// TwinCAT 3 PLC project TcComposite
// Title: TcComposite
// Company: Krystian Lis
// Author: Krystian Lis
// ProjectVersion: 0.001
// ProgramVersion: 3.1.4023.0
// libraries:
//   Tc2_Standard, * (Beckhoff Automation GmbH)
//   Tc2_System, * (Beckhoff Automation GmbH)
//   Tc2_Utilities, * (Beckhoff Automation GmbH)
//   Tc3_Module, * (Beckhoff Automation GmbH)
//   VisuDialogs, * (System)
// project tree:
//   DUTs/TestSt/ ST_PID.TcDUT
//   / GlobalTextList.TcGTLO, PlcTask.TcTTO, Visualization Manager.TcVMO (not stored), VISU_TASK.TcTTO
//   GVLs/ GVL_Data.TcGVL, G.TcGVL, GVL_Sys.TcGVL
//   POUs/Loggers/Functions/ F_Log.TcPOU, UINT_TO_ZEROSTRING.TcPOU
//   POUs/Loggers/ LogList.TcPOU
//   POUs/Objects/Abstracts/Base/ I_BoolPub.TcIO, I_BoolSub.TcIO
//   POUs/Objects/Abstracts/ I_Object.TcIO, I_SYS_COMP_Object.TcIO, Object.TcPOU
//   POUs/Objects/Base/ BoolSub.TcPOU, BoolPub.TcPOU
//   POUs/Objects/Composite/ Timer.TcPOU
//   POUs/Objects/ObjectList/Functions/ F_Get_Parent_Path.TcPOU
//   POUs/Objects/ObjectList/ _SYS_COMP_FirstObject.TcPOU, _SYS_COMP_.TcPOU
//   POUs/Objects/TestObj/ A.TcPOU, B.TcPOU, C.TcPOU
//   POUs/Params/Abstracts/ BaseParam.TcPOU, I_Param.TcIO
//   POUs/Params/ BoolParam.TcPOU, DintParam.TcPOU, RealParam.TcPOU, TimeParam.TcPOU, UdintParam.TcPOU
//   POUs/Params/Functions/ F_Change_Param.TcPOU, F_IObject_TO_IParam.TcPOU
//   POUs/Programs/ MAIN.TcPOU
//   POUs/System/Abstracts/ I_Blank.TcIO, I_Label.TcIO, Label.TcPOU
//   VISUs/ LandingPage.TcVIS, ObjectBrowser.TcVIS, ParamDialog.TcVIS, LogVisu.TcVIS, VisuComments.TcPOU
// real-time tasks:
//   TASK PlcTask: cycle T#10ms, priority 20, ADS port 350
//   TASK VISU_TASK: cycle T#200000us, priority 30, ADS port 351

CONFIGURATION TcComposite
    RESOURCE PLC ON TwinCAT3
        TASK PlcTask(INTERVAL := T#10ms, PRIORITY := 20);
        TASK VISU_TASK(INTERVAL := T#200000us, PRIORITY := 30);
        PROGRAM MAIN WITH PlcTask : MAIN;
        PROGRAM VisuElems_Visu_Prg WITH VISU_TASK : VisuElems.Visu_Prg;
    END_RESOURCE
END_CONFIGURATION

// ---- DUTs/TestSt/ST_PID.TcDUT
//Test structure
//Check if object can ignore struct types when trying to find its parent
// Parent
//	-Struct
//	--Child 1
//	--Child 2
//	--Child 3
//Struct should be ignored and child should be added directly to the parent


TYPE ST_PID :
STRUCT
	p: RealParam;
	i: RealParam;
	d: RealParam;
END_STRUCT
END_TYPE

// ---- GVLs/GVL_Data.TcGVL
//Test GVL
{attribute 'qualified_only'}
VAR_GLOBAL
END_VAR

// ---- GVLs/G.TcGVL
//Test GVL
{attribute 'qualified_only'}
VAR_GLOBAL
A1: A;
A2: A;
A3: A;
END_VAR

// ---- GVLs/GVL_Sys.TcGVL
//Test GVL
{attribute 'qualified_only'}
VAR_GLOBAL
END_VAR

// ---- POUs/Objects/Abstracts/Base/I_BoolPub.TcIO
INTERFACE I_BoolPub EXTENDS I_SYS_COMP_Object

//Work in progress

METHOD Attach_Sub
VAR_INPUT
	IObject: I_SYS_COMP_Object;
END_VAR
END_METHOD

PROPERTY Get : BOOL
GET
END_GET
END_PROPERTY

METHOD Remove_Sub
VAR_INPUT
	IObject: I_SYS_COMP_Object;
END_VAR
END_METHOD

END_INTERFACE

// ---- POUs/Objects/Abstracts/Base/I_BoolSub.TcIO
INTERFACE I_BoolSub EXTENDS I_SYS_COMP_Object

//Work in progress

METHOD Attach_Pub
VAR_INPUT
	IObject: I_SYS_COMP_Object;
END_VAR
END_METHOD

METHOD Remove_Pub
VAR_INPUT
	IObject: I_SYS_COMP_Object;
END_VAR
END_METHOD

PROPERTY Set : BOOL
SET
END_SET
END_PROPERTY

END_INTERFACE

// ---- POUs/Objects/Abstracts/I_Object.TcIO
INTERFACE I_Object EXTENDS I_Label

//I_SYS_COMP_Object facade

METHOD Get_Child : I_Object
VAR_INPUT
	name: STRING;
END_VAR
END_METHOD

METHOD Get_Parent : I_Object
VAR_INPUT
END_VAR
END_METHOD

METHOD Refresh
VAR_INPUT
END_VAR
END_METHOD

END_INTERFACE

// ---- POUs/Objects/Abstracts/I_SYS_COMP_Object.TcIO
INTERFACE I_SYS_COMP_Object EXTENDS I_Label

//System interface, shouldn't be modified

METHOD _SYS_COMP_Add_Child_
VAR_INPUT
	IObject: I_SYS_COMP_Object;
END_VAR
END_METHOD

METHOD _SYS_COMP_Get_Child : I_SYS_COMP_Object
VAR_INPUT
	name: STRING;
END_VAR
END_METHOD

METHOD _SYS_COMP_Get_Object : I_SYS_COMP_Object
VAR_INPUT
	parent_name: STRING;
	name: STRING;
END_VAR
END_METHOD

PROPERTY _SYS_COMP_last_child : I_SYS_COMP_Object
GET
END_GET
END_PROPERTY

PROPERTY _SYS_COMP_next_object : I_SYS_COMP_Object
GET
END_GET
SET
END_SET
END_PROPERTY

PROPERTY _SYS_COMP_parent : I_SYS_COMP_Object
GET
END_GET
SET
END_SET
END_PROPERTY

PROPERTY _SYS_COMP_prev_object : I_SYS_COMP_Object
GET
END_GET
SET
END_SET
END_PROPERTY

METHOD _SYS_COMP_Remove_Child_
VAR_INPUT
	IObject: I_SYS_COMP_Object;
END_VAR
END_METHOD

END_INTERFACE

// ---- POUs/Params/Abstracts/I_Param.TcIO
INTERFACE I_Param EXTENDS I_Label

METHOD Change_Param
VAR_INPUT
	value: STRING;
END_VAR
END_METHOD

PROPERTY display : STRING
GET
END_GET
END_PROPERTY

END_INTERFACE

// ---- POUs/System/Abstracts/I_Blank.TcIO
INTERFACE I_Blank EXTENDS __SYSTEM.IQueryInterface

END_INTERFACE

// ---- POUs/System/Abstracts/I_Label.TcIO
INTERFACE I_Label EXTENDS I_Blank

PROPERTY name : STRING
GET
END_GET
END_PROPERTY

END_INTERFACE

// ---- POUs/Programs/MAIN.TcPOU
PROGRAM MAIN
VAR
	rParam: I_Object;

	_init: BOOL;
END_VAR

IF NOT _init THEN
	
	F_Change_Param(
		G.A1.Get_Child('B1').Get_Child('tB'),
		'TRUE');
		
	rParam := G.A1.Get_Child('C1').Get_Child('tR');
	F_Change_Param(rParam, '0.7');

	
	_init := TRUE;
END_IF

END_PROGRAM

// ---- POUs/Params/Functions/F_Change_Param.TcPOU
FUNCTION F_Change_Param : BOOL
VAR_INPUT
	IObject: I_Object;
	value: STRING;
END_VAR
VAR
	_IParam: I_Param;
	_interface_match: BOOL;
END_VAR

//Used to safely change param of unknown object. If object doesn't contain I_Param
//or if it is 0 then it won't work.

_interface_match := __QUERYINTERFACE(IObject, _IParam);
IF _interface_match THEN
	_IParam.Change_Param(value);
END_IF

F_Change_Param := _interface_match;

END_FUNCTION

// ---- POUs/Objects/TestObj/A.TcPOU
{attribute 'call_after_init'}
FUNCTION_BLOCK A EXTENDS Object
VAR_INPUT
END_VAR
VAR_OUTPUT
END_VAR
VAR
	B1: B;
	B2: B;
	B3: B;

	tR: RealParam;
END_VAR

END_FUNCTION_BLOCK

// ---- POUs/Objects/Abstracts/Object.TcPOU
FUNCTION_BLOCK ABSTRACT Object EXTENDS Label IMPLEMENTS I_SYS_COMP_Object, I_Object
VAR

	{attribute 'no_copy'}
	{attribute 'no_init'}
	_SYS_COMP_next_object_: I_SYS_COMP_Object;
	
	{attribute 'no_copy'}
	{attribute 'no_init'}
	_SYS_COMP_prev_object_: I_SYS_COMP_Object;
	
	{attribute 'no_copy'}
	{attribute 'no_init'}
	_SYS_COMP_last_child_: I_SYS_COMP_Object;
	
	{attribute 'no_copy'}
	{attribute 'no_init'}
	_SYS_COMP_parent_: I_SYS_COMP_Object;
	
	{attribute 'no_copy'}
	{attribute 'no_init'}
	_SYS_COMP_init_parent_: BOOL;
	
END_VAR

METHOD _SYS_COMP_Add_Child_
VAR_INPUT
	IObject: I_SYS_COMP_Object;
END_VAR
//Remove from current chain and add to parent chain



IF IObject = 0 THEN
	RETURN;
END_IF

IF IObject._SYS_COMP_parent <> 0 THEN
	RETURN;
END_IF

//_SYS_COMP_.Remove_Object(IObject);

F_Log(IObject, 'ADDED TO', THIS^, '', 0);



IObject._SYS_COMP_parent := THIS^;



IF _SYS_COMP_last_child_ = 0 THEN
	_SYS_COMP_last_child_ := IObject;
	//LOG
	RETURN;	
END_IF


IObject._SYS_COMP_prev_object := _SYS_COMP_last_child_;

_SYS_COMP_last_child_._SYS_COMP_next_object := IObject;


_SYS_COMP_last_child_ := IObject;
END_METHOD

METHOD _SYS_COMP_Find_Parent_
VAR
	_temp_name: STRING;
	_potential_parent: I_SYS_COMP_Object;
END_VAR
// At the initialisation all objects are added to 
// the global list in order parent, child, parent_sibling, parent_sibling_child etc

// At FB_init the object is added to global list and then it's looking for parent
// It first check if previous sybling is its parent, 
// and then if its parent of a parent(of a parent ...)
// if there is no similarity beteen objec and any other object paths,
// the object is not removed from global list.

// Example child name: A.B.C.D.E
// Example previous sibling name: G.A.B
// Example parent name: G.A.B
//Thus the process looks like that:

IF _SYS_COMP_prev_object_ = 0 THEN
	RETURN;
END_IF

//Check if previous sybling has similar path as the object
IF FIND(_name, _SYS_COMP_prev_object_.name) <> 0 THEN
	_temp_name := F_Get_Parent_Path(_name);
	//delete name after last dot and check if it matches previous sybling name
	IF _SYS_COMP_prev_object_.name = _temp_name THEN
		_SYS_COMP_prev_object_._SYS_COMP_Add_Child_(THIS^);
		RETURN;
	END_IF
	
	//proceed deleting dots, if any name match the resulting path then set up the parent
	WHILE TRUE DO
		_temp_name := F_Get_Parent_Path(_temp_name);
		_potential_parent := _SYS_COMP_prev_object._SYS_COMP_Get_Child(_temp_name);

		IF _potential_parent <> _SYS_COMP_prev_object THEN
			_potential_parent._SYS_COMP_Add_Child_(THIS^);
			RETURN;	
		END_IF
		
		// if nothing left from the object path, then the object is part of global list
		IF _temp_name = '' THEN
			RETURN;
		END_IF
	END_WHILE
END_IF
END_METHOD

METHOD _SYS_COMP_Get_Child : I_SYS_COMP_Object
VAR_INPUT
	name: STRING;
END_VAR
VAR
	_IObject: I_SYS_COMP_Object;
END_VAR
//Get system object interface

//Add # at the end. This will ensure that the string value 
//is actually on the end of the path
IF RIGHT(name, 1) <> '#' THEN
	name := CONCAT(name, '#');
END_IF

IF _SYS_COMP_last_child_ <> 0 THEN
	_IObject := _SYS_COMP_last_child_._SYS_COMP_Get_Object(_name, name);
END_IF

//For security reasons this method always returns something,
//Thus if object can't be found, the methods return the THIS object
IF _IObject <> 0 THEN
	_SYS_COMP_Get_Child := _IObject;
ELSE
	_SYS_COMP_Get_Child := THIS^;
END_IF
END_METHOD

METHOD _SYS_COMP_Get_Object : I_SYS_COMP_Object
VAR_INPUT
	parent_name: STRING;
	name: STRING;
END_VAR
VAR
	_temp_name: STRING;
	_IObject: I_SYS_COMP_Object;
	_case: USINT;
END_VAR
_temp_name := CONCAT(_name, '#');

IF parent_name = '#' THEN
	//FIND object ending with name# in any parent
	_case := 1;
END_IF

//Check if object matches the searched name,
//If no check if it contain searched name,
//If yes, check in children,
//If not, go to next sibling

CASE _case OF
	0:
		IF FIND(_temp_name, name) <> 0 THEN
			_SYS_COMP_Get_Object := THIS^;
			RETURN;
		END_IF
		IF FIND(_temp_name, parent_name) <> 0 THEN
			_IObject := _SYS_COMP_Get_Child(name);
			IF _IObject <> 0 AND_THEN _name <> _IObject.name THEN
				_SYS_COMP_Get_Object := _IObject;
				RETURN;
			END_IF
		END_IF
	1:	//FIND object ending with name# in any parent
		IF FIND(_temp_name, name) <> 0 THEN
			_SYS_COMP_Get_Object := THIS^;
			RETURN;	
		ELSE
			_IObject := _SYS_COMP_Get_Child(name);
			IF _IObject <> 0 AND_THEN _name <> _IObject.name THEN
				_SYS_COMP_Get_Object := _IObject;
				RETURN;
			END_IF
		END_IF
END_CASE


//Got to next sibling
IF _SYS_COMP_prev_object_ <> 0 THEN
	_SYS_COMP_Get_Object := _SYS_COMP_prev_object_._SYS_COMP_Get_Object(parent_name, name);
	RETURN;
END_IF
END_METHOD

PROPERTY _SYS_COMP_last_child : I_SYS_COMP_Object
GET
_SYS_COMP_last_child := _SYS_COMP_last_child_;
END_GET
END_PROPERTY

PROPERTY _SYS_COMP_next_object : I_SYS_COMP_Object
GET
_SYS_COMP_next_object := _SYS_COMP_next_object_;
END_GET
SET
//F_Log(THIS^, 'ATTACH_NEXT', next_object, 'BEFORE', _next_object);
_SYS_COMP_next_object_ := _SYS_COMP_next_object;
END_SET
END_PROPERTY

PROPERTY _SYS_COMP_parent : I_SYS_COMP_Object
GET
_SYS_COMP_parent := _SYS_COMP_parent_;
END_GET
SET
IF NOT _SYS_COMP_init_parent_ THEN
	_SYS_COMP_parent_ := _SYS_COMP_parent;
	_SYS_COMP_init_parent_ := TRUE;
END_IF
END_SET
END_PROPERTY

PROPERTY _SYS_COMP_prev_object : I_SYS_COMP_Object
GET
_SYS_COMP_prev_object := _SYS_COMP_prev_object_;
END_GET
SET
//F_Log(THIS^, 'ATTACH_PREV', prev_object, 'BEFORE', _prev_object);
_SYS_COMP_prev_object_ := _SYS_COMP_prev_object;
END_SET
END_PROPERTY

METHOD _SYS_COMP_Remove_Child_
VAR_INPUT
	IObject: I_SYS_COMP_Object;
END_VAR
IF IObject = 0 THEN
	//LOG
	RETURN;
END_IF

IF _SYS_COMP_last_child_ = 0 THEN
	//LOG
	RETURN;
END_IF

IF IObject._SYS_COMP_parent <> 0 AND_THEN IObject._SYS_COMP_parent.name <> _name THEN
	//LOG
	//Object from different parent
	F_Log(IObject, 'IS NOT CHILD OF', THIS^, '', 0);
	RETURN;
END_IF

F_Log(IObject, 'REMOVED FROM', THIS^, '', 0);

IF IObject._SYS_COMP_next_object = 0 AND IObject._SYS_COMP_prev_object <> 0 THEN
	_SYS_COMP_last_child_ := IObject._SYS_COMP_prev_object;
	_SYS_COMP_last_child_._SYS_COMP_next_object := 0;
	
	_SYS_COMP_last_child_ := 0;
	IObject._SYS_COMP_next_object := 0;
	IObject._SYS_COMP_prev_object := 0;
	//LOG
	RETURN;
END_IF

IF IObject._SYS_COMP_next_object <> 0 AND IObject._SYS_COMP_prev_object <> 0 THEN
	IObject._SYS_COMP_next_object._SYS_COMP_prev_object := IObject._SYS_COMP_prev_object;
	IObject._SYS_COMP_prev_object._SYS_COMP_next_object := IObject._SYS_COMP_next_object;


	IObject._SYS_COMP_next_object := 0;
	IObject._SYS_COMP_prev_object := 0;
	//LOG
	RETURN;
END_IF

IF IObject._SYS_COMP_next_object <> 0 AND IObject._SYS_COMP_prev_object = 0 THEN
	IObject._SYS_COMP_next_object._SYS_COMP_prev_object := 0;

	IObject._SYS_COMP_next_object := 0;
	IObject._SYS_COMP_prev_object := 0;
	//LOG
	RETURN;
END_IF
END_METHOD

METHOD FB_exit : BOOL
VAR_INPUT
	bInCopyCode : BOOL; // if TRUE, the exit method is called for exiting an instance that is copied afterwards (online change).
END_VAR
//_SYS_COMP_.Remove_Object(THIS^);
END_METHOD

METHOD FB_init : BOOL
VAR_INPUT
	bInitRetains : BOOL; // if TRUE, the retain variables are initialized (warm start / cold start)
	bInCopyCode : BOOL;  // if TRUE, the instance afterwards gets moved into the copy code (online change)
END_VAR
_SYS_COMP_.Add_Object(THIS^);
_SYS_COMP_Find_Parent_();
END_METHOD

METHOD Get_Child : I_Object
VAR_INPUT
	name: STRING;
END_VAR
VAR
	IChild: I_Object;
	ISYSChild: I_SYS_COMP_Object;
END_VAR
//Get child facade interface(without all system methods)

ISYSChild := _SYS_COMP_Get_Child(name);

IF __QUERYINTERFACE(ISYSChild, IChild) THEN
	Get_Child := IChild;
ELSE
	Get_Child := THIS^;
END_IF
END_METHOD

METHOD Get_Parent : I_Object
VAR
	IParent : I_Object;
END_VAR
//Get parent facade interface(without all system methods)

IF __QUERYINTERFACE(_SYS_COMP_parent_, IParent) THEN
	Get_Parent := IParent;
ELSE
	Get_Parent := THIS^;
END_IF
END_METHOD

METHOD Refresh
VAR_INPUT
END_VAR
//User code. Called by children
END_METHOD

END_FUNCTION_BLOCK

// ---- POUs/System/Abstracts/Label.TcPOU
{attribute 'reflection'}
FUNCTION_BLOCK ABSTRACT Label IMPLEMENTS I_Label
VAR CONSTANT
END_VAR
VAR_INPUT
END_VAR
VAR
	
	{attribute 'instance-path'} 
    {attribute 'noinit'}
	_sPath: T_MaxString;
	{attribute 'no_copy'}
	_name: T_MaxString;
	
END_VAR

//Base class. Allows to querry instances by their name.

METHOD FB_init : BOOL
VAR_INPUT
	bInitRetains : BOOL; // if TRUE, the retain variables are initialized (warm start / cold start)
	bInCopyCode : BOOL;  // if TRUE, the instance afterwards gets moved into the copy code (online change)
END_VAR
//Update name after each 'New Download'
_name := DELETE(_sPath, FIND(_sPath, '.'), 1);
_name := DELETE(_name, FIND(_name, '.'), 1);
END_METHOD

PROPERTY name : STRING
GET
name := _name;
END_GET
END_PROPERTY

END_FUNCTION_BLOCK

// ---- POUs/Loggers/Functions/F_Log.TcPOU
FUNCTION F_Log : BOOL
VAR_INPUT
	obj_1	: I_SYS_COMP_Object;
	act_1	: STRING(30);
	obj_2	: I_SYS_COMP_Object;
	act_2	: STRING(30);
	obj_3	: I_SYS_COMP_Object;
END_VAR
VAR
	_remaining_spaces: INT;
	_temp_string: T_MAXSTRING := '                                                                                                                                                                                                                                                               ';
	
	_obj_1_name	: STRING(65);
	_obj_2_name	: STRING(65);
	_obj_3_name	: STRING(65);

END_VAR

//This function creates logs regarding any system related events such as
//Add/Remove Child/Parent etc.

IF obj_1 <> 0 THEN
	_obj_1_name := obj_1.name;
END_IF
IF obj_2 <> 0 THEN
	_obj_2_name := obj_2.name;
END_IF
IF obj_3 <> 0 THEN
	_obj_3_name := obj_3.name;
END_IF

_temp_string := INSERT(_temp_string, _obj_1_name, 0);
_temp_string := INSERT(_temp_string, act_1, 64);
_temp_string := INSERT(_temp_string, _obj_2_name, 94);
_temp_string := INSERT(_temp_string, act_2, 159);
_temp_string := INSERT(_temp_string, _obj_3_name, 189);

LogList.AddLog(_temp_string);

END_FUNCTION

// ---- POUs/Loggers/LogList.TcPOU
{attribute 'global_init_slot' := '40001'}
PROGRAM LogList
VAR
	list: ARRAY[1..4000] OF T_MAXSTRING;
	lastlog: UINT := 1;
END_VAR

//Singleton containing logs

METHOD AddLog
VAR_INPUT
	text: T_MAXSTRING;
END_VAR
list[lastLog] := text;
lastLog := lastLog + 1;

IF lastLog = 4001 THEN
	lastLog := 1;
END_IF
END_METHOD

METHOD Print_To_ADS : DINT
VAR
	_counter : UINT := 1;
	_temp_string: T_MAXSTRING;
	_print_string: T_MAXSTRING;
	_error : DINT;
END_VAR
FOR _counter := 1 TO lastlog DO
	_temp_string := UINT_TO_ZEROSTRING(_counter);
	_temp_string := CONCAT(_temp_string, '  ');
	_temp_string := CONCAT(_temp_string, list[_counter]);
	_print_string := _temp_string;
	
	_error := ADSLOGSTR(ADSLOG_MSGTYPE_STRING, _print_string, '');
	
	IF _error <> 0 THEN
		Print_To_ADS := _error;
		RETURN;
	END_IF
END_FOR
END_METHOD

END_PROGRAM

// ---- POUs/Loggers/Functions/UINT_TO_ZEROSTRING.TcPOU
FUNCTION UINT_TO_ZEROSTRING : T_MAXSTRING
VAR_INPUT
	input : UDINT;
END_VAR
VAR
	tempString : T_MAXSTRING;
END_VAR

tempString := TO_STRING(input);
WHILE LEN(tempString) < 4 DO
	tempString := INSERT(tempString, '0', 0);
END_WHILE
UINT_TO_ZEROSTRING := tempString;

END_FUNCTION

// ---- POUs/Objects/ObjectList/Functions/F_Get_Parent_Path.TcPOU
FUNCTION F_Get_Parent_Path : T_MAXSTRING
VAR_INPUT
	child_path: T_MAXSTRING;
END_VAR
VAR
	_output_string: T_MAXSTRING;
	_dot_position: INT;
END_VAR

WHILE TRUE DO
	_dot_position := FIND(child_path, '.');	
	
	IF _dot_position = 0 THEN
		_output_string := DELETE(_output_string, 1, LEN(_output_string));
		F_Get_Parent_Path := _output_string;
		RETURN;
	END_IF
	
	_output_string := CONCAT(_output_string, LEFT(child_path, _dot_position));
		
	child_path := DELETE(child_path, _dot_position, 1);
	

END_WHILE

END_FUNCTION

// ---- POUs/Objects/ObjectList/_SYS_COMP_.TcPOU
{attribute 'global_init_slot' := '40002'}
{attribute 'hide_all_locals'}
PROGRAM _SYS_COMP_
VAR
	_last_in_chain: I_SYS_COMP_Object;
	_object_list: _SYS_COMP_FirstObject;
END_VAR
VAR CONSTANT
	_name : STRING := 'ObjectList';
END_VAR

METHOD Add_Object
VAR_INPUT
	IObject: I_SYS_COMP_Object;
END_VAR
IF IObject = 0 THEN
	//LOG
	RETURN;
END_IF

//Remove_Object(IObject);

F_Log(IObject, 'ADDED TO', _object_list, '', 0);

IF _last_in_chain = 0 THEN
	_last_in_chain := IObject;
	RETURN;
END_IF

_last_in_chain._SYS_COMP_next_object := IObject;
IObject._SYS_COMP_prev_object := _last_in_chain;
_last_in_chain := IObject;
END_METHOD

METHOD Get_Object : I_SYS_COMP_Object
VAR_INPUT
	name: STRING;
END_VAR
VAR
	_IObject	:	I_SYS_COMP_Object;
END_VAR
name := CONCAT(name, '#');
IF _last_in_chain <> 0 THEN
	_IObject := _last_in_chain._SYS_COMP_Get_Object('#', name);
END_IF

IF _IObject <> 0 THEN
	Get_Object := _IObject;
ELSE
	Get_Object := _object_list;
END_IF

//LOG
END_METHOD

PROPERTY object_list : I_SYS_COMP_Object
GET
object_list := _object_list;
END_GET
END_PROPERTY

METHOD Remove_Object
VAR_INPUT
	IObject: I_SYS_COMP_Object;
END_VAR
IF IObject = 0 THEN
	RETURN;
END_IF

IF IObject._SYS_COMP_prev_object = 0 AND IObject._SYS_COMP_next_object = 0 THEN
	RETURN;
END_IF

IF IObject._SYS_COMP_parent <> 0 THEN
	IObject._SYS_COMP_parent._SYS_COMP_Remove_Child_(IObject);
	RETURN;
END_IF

F_Log(IObject, 'REMOVED FROM', _object_list, '', 0);

IF IObject._SYS_COMP_next_object <> 0 AND IObject._SYS_COMP_prev_object <> 0 THEN
	IObject._SYS_COMP_next_object._SYS_COMP_prev_object := IObject._SYS_COMP_prev_object;
	IObject._SYS_COMP_prev_object._SYS_COMP_next_object := IObject._SYS_COMP_next_object;
	
	IObject._SYS_COMP_next_object := 0;
	IObject._SYS_COMP_prev_object := 0;
	
	
	RETURN;
END_IF

IF IObject._SYS_COMP_next_object = 0 AND IObject._SYS_COMP_prev_object <> 0 THEN
	IObject._SYS_COMP_prev_object._SYS_COMP_next_object := 0;
	_last_in_chain := IObject._SYS_COMP_prev_object;
	
	IObject._SYS_COMP_next_object := 0;
	IObject._SYS_COMP_prev_object := 0;

	RETURN;
END_IF

IF IObject._SYS_COMP_next_object <> 0 AND IObject._SYS_COMP_prev_object = 0 THEN
	IObject._SYS_COMP_next_object._SYS_COMP_prev_object := 0;
	
	IObject._SYS_COMP_next_object := 0;
	IObject._SYS_COMP_prev_object := 0;
	
	RETURN;
END_IF

//LOG
END_METHOD

END_PROGRAM

// ---- POUs/Objects/ObjectList/_SYS_COMP_FirstObject.TcPOU
{attribute 'call_after_init'}
FUNCTION_BLOCK FINAL _SYS_COMP_FirstObject EXTENDS Object
VAR_INPUT
END_VAR
VAR_OUTPUT
END_VAR
VAR
END_VAR

//First object in global object list.
//DO NOT DELETE!!!

END_FUNCTION_BLOCK

// ---- POUs/Objects/TestObj/B.TcPOU
{attribute 'call_after_init'}
FUNCTION_BLOCK B EXTENDS Object
VAR_INPUT
END_VAR
VAR_OUTPUT
END_VAR
VAR
	C1: C;
	C2: C;
	C3: C;

	tR: RealParam;
END_VAR

END_FUNCTION_BLOCK

// ---- POUs/Objects/TestObj/C.TcPOU
{attribute 'call_after_init'}
FUNCTION_BLOCK C EXTENDS Object
VAR_INPUT
END_VAR
VAR_OUTPUT
END_VAR
VAR
	tU: UdintParam;
	tT: TimeParam;
	tR: RealParam;
END_VAR

END_FUNCTION_BLOCK

// ---- POUs/Params/UdintParam.TcPOU
{attribute 'call_after_init'}
FUNCTION_BLOCK FINAL UdintParam EXTENDS BaseParam
VAR_INPUT
END_VAR
VAR_OUTPUT
	value: UDINT;
END_VAR
VAR
	
END_VAR

METHOD Change_Param
VAR_INPUT
	value	: STRING;
END_VAR
THIS^.value := STRING_TO_UDINT(value);
_display := UDINT_TO_STRING(THIS^.value);
END_METHOD

METHOD Quick_Change
VAR_INPUT
	value: UDINT;
END_VAR
THIS^.value := value;
_display := UDINT_TO_STRING(THIS^.value);
END_METHOD

END_FUNCTION_BLOCK

// ---- POUs/Params/Abstracts/BaseParam.TcPOU
FUNCTION_BLOCK ABSTRACT BaseParam EXTENDS Object IMPLEMENTS I_Param
VAR
	_display: STRING := '0';
END_VAR

//Base Param object.
// _display should be used to extract data from the interface in string form. 
// For example to use with visu.

//Q variable should be used to access the data directly from FB.
//Each derivative of this funciton should have added Q variable of literal type.

//Each derivative of BaseParam has Quick_Change(value) to directly modify Q value.

METHOD Change_Param
VAR_INPUT
	value	: STRING;
END_VAR
//How string value should be translated to other data type
END_METHOD

PROPERTY display : STRING
GET
display := _display;
END_GET
END_PROPERTY

END_FUNCTION_BLOCK

// ---- POUs/Params/TimeParam.TcPOU
{attribute 'call_after_init'}
FUNCTION_BLOCK FINAL TimeParam EXTENDS BaseParam
VAR_INPUT
END_VAR
VAR_OUTPUT
	value: TIME;
END_VAR
VAR
END_VAR

METHOD Change_Param
VAR_INPUT
	value	: STRING;
END_VAR
VAR
	_last_char: STRING;
	_value_ms: DWORD;
END_VAR
//This method changes the TIME value. It accepts more TIME formats than standard T#12s.
//Accepted formats include:
// - 12s, 12S, 12 s, 12 S, T#12S, T#12s, T#0m12S, 12000, etc

value := F_ToLCase(value);

WHILE FIND(value, ' ') <> 0 DO
	value := DELETE(value, 1, FIND(value, ' '));
END_WHILE

_last_char := RIGHT(value, 1);
IF _last_char <> 's' AND _last_char <> 'm' AND _last_char <> 'h' AND _last_char <> 'd' THEN
	_value_ms := STRING_TO_DWORD(value);
	value := DWORD_TO_STRING(_value_ms);
	value := concat(value, 'ms');
END_IF

value := DELETE(value, 1, FIND(value, 't#'));
value := CONCAT('T#', value);

THIS^.value := STRING_TO_TIME(value);
_display := TIME_TO_STRING(THIS^.value);
_display := DELETE(_display, 2, 1);
END_METHOD

METHOD Quick_Change
VAR_INPUT
	value: TIME;
END_VAR
THIS^.value := value;
_display := TIME_TO_STRING(THIS^.value);
_display := DELETE(_display, 2, 1);
END_METHOD

END_FUNCTION_BLOCK

// ---- POUs/Params/RealParam.TcPOU
{attribute 'call_after_init'}
FUNCTION_BLOCK FINAL RealParam EXTENDS BaseParam
VAR_INPUT
END_VAR
VAR_OUTPUT
	value: REAL;
END_VAR
VAR
	
END_VAR

METHOD Change_Param
VAR_INPUT
	value	: STRING;
END_VAR
THIS^.value := STRING_TO_REAL(value);
_display := REAL_TO_STRING(THIS^.value);
END_METHOD

METHOD Quick_Change
VAR_INPUT
	value: REAL;
END_VAR
THIS^.value := value;
_display := REAL_TO_STRING(THIS^.value);
END_METHOD

END_FUNCTION_BLOCK

// ---- POUs/Objects/Base/BoolSub.TcPOU
FUNCTION_BLOCK BoolSub EXTENDS Object IMPLEMENTS I_BoolSub
VAR_OUTPUT
	Q: BOOL;
END_VAR
VAR
	_pub: I_BoolPub;
END_VAR

//Work in progress

METHOD Attach_Pub
VAR_INPUT
	IObject: I_SYS_COMP_Object;
END_VAR
VAR
	_pub: I_BoolPub;
END_VAR
END_METHOD

METHOD Remove_Pub
VAR_INPUT
	IObject: I_SYS_COMP_Object;
END_VAR
VAR
	_pub: I_BoolPub;
END_VAR
END_METHOD

PROPERTY Set : I_SYS_COMP_Object
SET
Q := Set;
END_SET
END_PROPERTY

END_FUNCTION_BLOCK

// ---- POUs/Objects/Base/BoolPub.TcPOU
FUNCTION_BLOCK BoolPub EXTENDS Object IMPLEMENTS I_BoolSub
VAR_INPUT
	IN: BOOL;
END_VAR
VAR
	_sub: I_BoolSub;
END_VAR

//Work in progress

METHOD Attach_Sub
VAR_INPUT
	IObject: I_SYS_COMP_Object;
END_VAR
VAR
	_ISub: I_BoolSub;
END_VAR
IF __QUERYINTERFACE(IObject, _ISub) THEN
	_sub := _ISub;
END_IF
END_METHOD

PROPERTY Get : I_SYS_COMP_Object
GET
IN := Get;
END_GET
END_PROPERTY

METHOD Remove_Sub
VAR_INPUT
	IObject: I_SYS_COMP_Object;
END_VAR
VAR
	_ISub: I_BoolSub;
END_VAR
IF __QUERYINTERFACE(IObject, _ISub) THEN
	_sub := _ISub;
END_IF
END_METHOD

END_FUNCTION_BLOCK

// ---- POUs/Objects/Composite/Timer.TcPOU
FUNCTION_BLOCK Timer EXTENDS Object
VAR_INPUT
END_VAR
VAR_OUTPUT
END_VAR
VAR
	_in: I_BoolSub;
	_q: I_BoolPub;
END_VAR

//Work in progress

METHOD Refresh
VAR_INPUT
END_VAR
END_METHOD

END_FUNCTION_BLOCK

// ---- POUs/Params/BoolParam.TcPOU
{attribute 'call_after_init'}
FUNCTION_BLOCK FINAL BoolParam EXTENDS BaseParam
VAR_INPUT
END_VAR
VAR_OUTPUT
	value: BOOL;
END_VAR
VAR
END_VAR

METHOD Change_Param
VAR_INPUT
	value	: STRING;
END_VAR
//Change value to TRUE or FALSE. By default Twincat accept only 'FALSE' as actual FALSE
//This methods extends number of strings that are considered as FALSE.


value := F_ToUCase(value);

IF value = '' OR value = '0' OR value = 'F' OR value = 'FALSE' OR value = 'OFF' THEN
	value := 'FALSE';
ELSE
	value := 'TRUE';
END_IF

THIS^.value := STRING_TO_BOOL(value);

IF THIS^.value THEN
	_display := 'ON';
ELSE
	_display := 'OFF';
END_IF
END_METHOD

METHOD Quick_Change
VAR_INPUT
	value: BOOL;
END_VAR
THIS^.value := value;

IF THIS^.value THEN
	_display := 'ON';
ELSE
	_display := 'OFF';
END_IF
END_METHOD

END_FUNCTION_BLOCK

// ---- POUs/Params/DintParam.TcPOU
{attribute 'call_after_init'}
FUNCTION_BLOCK FINAL DintParam EXTENDS BaseParam
VAR_INPUT
END_VAR
VAR_OUTPUT
	value: DINT;
END_VAR
VAR
	
END_VAR

METHOD Change_Param
VAR_INPUT
	value	: STRING;
END_VAR
THIS^.value := STRING_TO_DINT(value);
_display := DINT_TO_STRING(THIS^.value);
END_METHOD

METHOD Quick_Change
VAR_INPUT
	value: DINT;
END_VAR
THIS^.value := value;
_display := DINT_TO_STRING(THIS^.value);
END_METHOD

END_FUNCTION_BLOCK

// ---- POUs/Params/Functions/F_IObject_TO_IParam.TcPOU
FUNCTION F_IObject_TO_IParam : I_Param
VAR_INPUT
	IObject: I_SYS_COMP_Object;
	IParam: I_Param;
END_VAR
VAR
END_VAR

__QUERYINTERFACE(IObject, IParam);
F_IObject_To_IParam := IParam;

END_FUNCTION

// ---- VISUs/VisuComments.TcPOU
PROGRAM VisuComments
VAR
END_VAR

(*
//Visu consist of 2 frames:
	- Object browser	- used for browsing the object tree. It is possible to access every
						object through it. Side buttons are used to move between syblings.
						Buttons above and below current object name help to move between generations.
						Enter the name of the object on the middle and clikc 'Search' to find any object.
						
						- 'Change param' opens dialog that can be used to modify internal value of any object
						implementing I_Param interface. Use 'Copy Param from browser' each time the value or active object changed.
	
	- Logs				- contain all events, such as add or remove child, attach sub/pub, update sub, etc.


*)

END_PROGRAM

// ---- GlobalTextList.TcGTLO
TEXTLIST GlobalTextList
  253 = '%i'
  388 = '%s'
  847 = '<'
  19 = '< object'
  193 = '<<'
  317 = '<Previous Object'
  931 = '<Q'
  166 = '>'
  311 = '>>'
  81 = '>|'
  828 = 'Actions'
  34 = 'Actions:'
  105 = 'Change'
  414 = 'Change Param'
  201 = 'child'
  671 = 'Child'
  961 = 'Copy Object from browser'
  984 = 'Copy param from browser'
  895 = 'Copy Param from browser'
  293 = 'E>'
  609 = 'Enter'
  18 = 'Exit'
  571 = 'EXIT'
  239 = 'Get Last'
  350 = 'Get List'
  804 = 'Init'
  818 = 'Name'
  897 = 'Next Object'
  106 = 'object >'
  396 = 'Object Browser'
  15 = 'Parameter Browser'
  500 = 'parent'
  142 = 'Parent'
  957 = "Parent's Name:"
  108 = 'parent>'
  691 = 'Parents Name:'
  720 = 'Previous Object'
  669 = 'Refresh'
  852 = 'Search'
  892 = '^parent^'
  47 = '|<'
END_TEXTLIST

// ---- VISUs/LandingPage.TcVIS
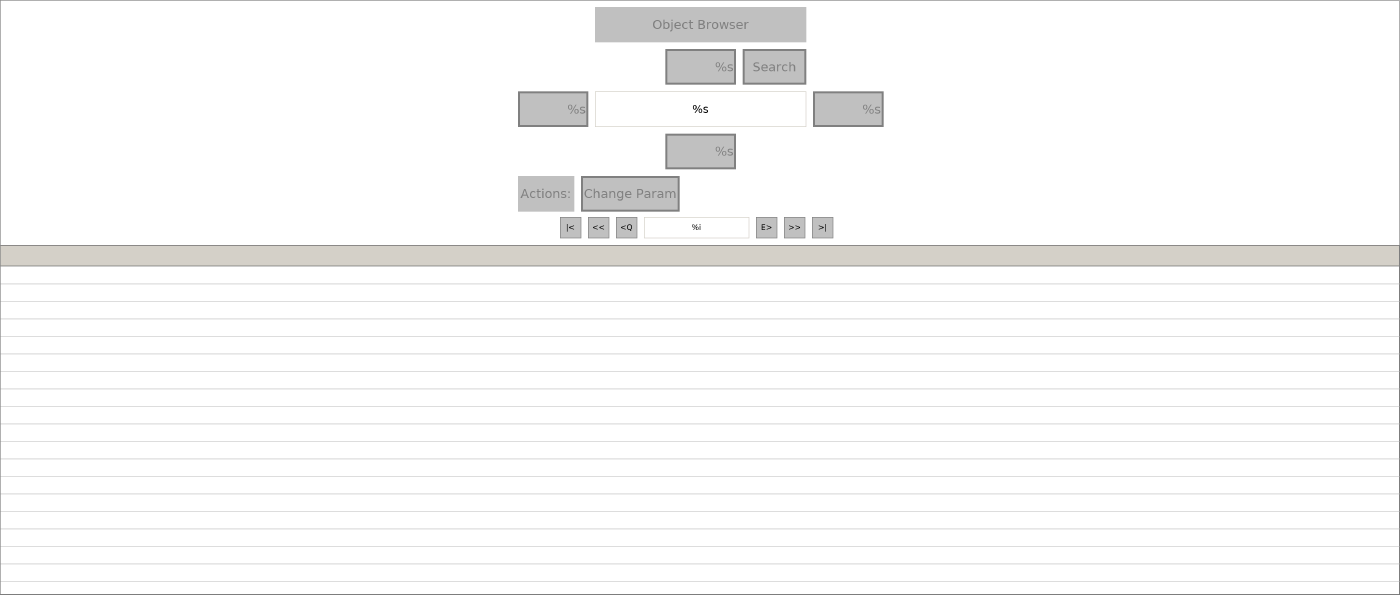
VISUALIZATION LandingPage  // 2000x850
    Frame (0,310 2000x540)
        shows LogVisu()
    Frame (730,0 532x302)
        shows ObjectBrowser()
END_VISUALIZATION

// ---- VISUs/ObjectBrowser.TcVIS
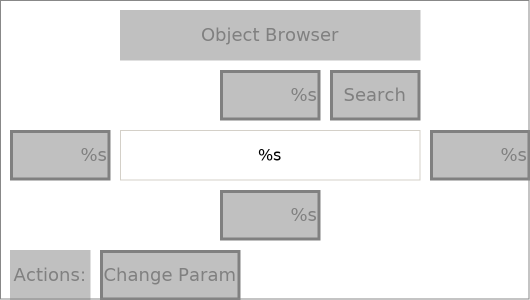
VISUALIZATION ObjectBrowser  // 530x300
VAR
	active_object: I_SYS_COMP_Object := _SYS_COMP_.object_list;
	
	search_name: STRING := 'Object';
	
	parent_name: STRING := '';
	child_name: STRING := '';
	
	next_object_name: STRING := '';
	prev_object_name: STRING := '';
	
END_VAR
    RoundedRectangle (120,10 300x50), "Object Browser"
    RoundedRectangle (10,130 100x50), "%s", text variable: CONCAT(prev_object_name, ' .')
        OnMouseUp: execute {
            IF active_object <> 0 AND_THEN active_object._SYS_COMP_prev_object <> 0 THEN
            	active_object := active_object._SYS_COMP_prev_object;
            	search_name := active_object.name;
            	IF active_object._SYS_COMP_parent <> 0 THEN
            		parent_name := active_object._SYS_COMP_parent.name;
            	ELSE
            		parent_name := 'Global Object.list';
            	END_IF
            	IF active_object._SYS_COMP_last_child <> 0 THEN
            		child_name := active_object._SYS_COMP_last_child.name;
            	ELSE
            		child_name := '';
            	END_IF
            	IF active_object._SYS_COMP_next_object <> 0 THEN
            		next_object_name := active_object._SYS_COMP_next_object.name;
            	ELSE
            		next_object_name := '';
            	END_IF
            	IF active_object._SYS_COMP_prev_object <> 0 THEN
            		prev_object_name := active_object._SYS_COMP_prev_object.name;
            	ELSE
            		prev_object_name := '';
            	END_IF
            END_IF
        }
    RoundedRectangle (430,130 100x50), "%s", text variable: CONCAT(next_object_name, ' .')
        OnMouseUp: execute {
            IF active_object <> 0 AND_THEN active_object._SYS_COMP_next_object <> 0 THEN
            	active_object := active_object._SYS_COMP_next_object;
            	search_name := active_object.name;
            	IF active_object._SYS_COMP_parent <> 0 THEN
            		parent_name := active_object._SYS_COMP_parent.name;
            	ELSE
            		parent_name := 'Global ObjectList';
            	END_IF
            	IF active_object._SYS_COMP_last_child <> 0 THEN
            		child_name := active_object._SYS_COMP_last_child.name;
            	ELSE
            		child_name := '';
            	END_IF
            	IF active_object._SYS_COMP_next_object <> 0 THEN
            		next_object_name := active_object._SYS_COMP_next_object.name;
            	ELSE
            		next_object_name := '';
            	END_IF
            	IF active_object._SYS_COMP_prev_object <> 0 THEN
            		prev_object_name := active_object._SYS_COMP_prev_object.name;
            	ELSE
            		prev_object_name := '';
            	END_IF
            END_IF
        }
    RoundedRectangle (220,190 100x50), "%s", text variable: CONCAT(child_name, ' .')
        OnMouseUp: execute {
            IF active_object <> 0 AND_THEN active_object._SYS_COMP_last_child <> 0 THEN
            	active_object := active_object._SYS_COMP_last_child;
            	search_name := active_object.name;
            	IF active_object._SYS_COMP_parent <> 0 THEN
            		parent_name := active_object._SYS_COMP_parent.name;
            	ELSE
            		parent_name := 'Global ObjectList';
            	END_IF
            	IF active_object._SYS_COMP_last_child <> 0 THEN
            		child_name := active_object._SYS_COMP_last_child.name;
            	ELSE
            		child_name := '';
            	END_IF
            	IF active_object._SYS_COMP_next_object <> 0 THEN
            		next_object_name := active_object._SYS_COMP_next_object.name;
            	ELSE
            		next_object_name := '';
            	END_IF
            	IF active_object._SYS_COMP_prev_object <> 0 THEN
            		prev_object_name := active_object._SYS_COMP_prev_object.name;
            	ELSE
            		prev_object_name := '';
            	END_IF
            END_IF
        }
    RoundedRectangle (220,70 100x50), "%s", text variable: CONCAT(parent_name, ' .')
        OnMouseUp: execute {
            IF active_object <> 0 AND_THEN active_object._SYS_COMP_parent <> 0 THEN
            	active_object := active_object._SYS_COMP_parent;
            	search_name := active_object.name;
            	IF active_object._SYS_COMP_parent <> 0 THEN
            		parent_name := active_object._SYS_COMP_parent.name;
            	ELSE
            		parent_name := 'Global ObjectList';
            	END_IF
            	IF active_object._SYS_COMP_last_child <> 0 THEN
            		child_name := active_object._SYS_COMP_last_child.name;
            	ELSE
            		child_name := '';
            	END_IF
            	IF active_object._SYS_COMP_next_object <> 0 THEN
            		next_object_name := active_object._SYS_COMP_next_object.name;
            	ELSE
            		next_object_name := '';
            	END_IF
            	IF active_object._SYS_COMP_prev_object <> 0 THEN
            		prev_object_name := active_object._SYS_COMP_prev_object.name;
            	ELSE
            		prev_object_name := '';
            	END_IF
            END_IF
        }
    Textfield (120,130 300x50), "%s", text variable: search_name
        OnMouseUp: write the text variable via Default
    RoundedRectangle (10,250 80x50), "Actions:"
    RoundedRectangle (100,250 140x50), "Change Param"
        OnMouseUp: OpenDialog Dialog=ParamDialog, Parameters={active_object: active_object, active_param: , name: , new_value: , value: }, OpenModal=True, OpenCentered=True
    RoundedRectangle (330,70 90x50), "Search"
        OnMouseUp: execute {
            active_object := _SYS_COMP_.Get_object(search_name);
            IF active_object <> 0 THEN
            	search_name := active_object.name;
            	IF active_object._SYS_COMP_parent <> 0 THEN
            		parent_name := active_object._SYS_COMP_parent.name;
            	ELSE
            		parent_name := 'Global ObjectList';
            	END_IF
            	IF active_object._SYS_COMP_last_child <> 0 THEN
            		child_name := active_object._SYS_COMP_last_child.name;
            	ELSE
            		child_name := '';
            	END_IF
            	IF active_object._SYS_COMP_next_object <> 0 THEN
            		next_object_name := active_object._SYS_COMP_next_object.name;
            	ELSE
            		next_object_name := '';
            	END_IF
            	IF active_object._SYS_COMP_prev_object <> 0 THEN
            		prev_object_name := active_object._SYS_COMP_prev_object.name;
            	ELSE
            		prev_object_name := '';
            	END_IF
            ELSE
            	search_name := 'OBJECT DOESNT EXIST';
            	parent_name := '';
            	child_name := '';
            	next_object_name := '';
            	prev_object_name := '';
            END_IF
        }
END_VISUALIZATION

// ---- VISUs/ParamDialog.TcVIS
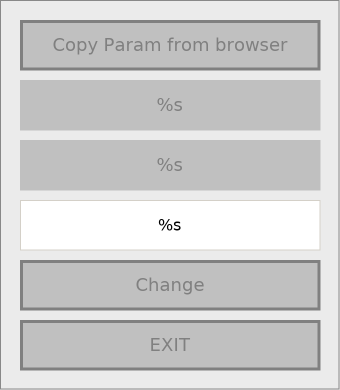
VISUALIZATION ParamDialog  // 340x390
VAR_INPUT
	active_object: I_SYS_COMP_Object;
END_VAR
VAR
	active_param: I_Param;
	name: STRING := 'ParamName';
	value: STRING := 'EnterNewValue';
	actual_value: STRING := 'ParamValue';

END_VAR
    RoundedRectangle (0,0 340x390)
    RoundedRectangle (20,140 300x50), "%s", text variable: actual_value
    RoundedRectangle (20,320 300x50), "EXIT"
        OnMouseUp: CloseDialog Dialog=ParamDialog, Result=OK, NumpadKeypadSet=True
    RoundedRectangle (20,20 300x50), "Copy Param from browser"
        OnMouseUp: execute {
            IF active_object <> 0 THEN
            	active_param := F_IObject_TO_IParam(active_object, active_param);
            	IF active_param <> 0 THEN
            		name := active_param.name;
            		value := active_param.display;
            		actual_value := active_param.display;
            	ELSE
            		name := 'Object is not Param!';
            		value := '';
            		actual_value := '';
            	END_IF
            ELSE
            	name := 'No Object selected!';
            	value := '';
            	actual_value := '';
            END_IF
        }
    Textfield (20,200 300x50), "%s", text variable: value
        OnMouseUp: write the text variable via Default
    RoundedRectangle (20,260 300x50), "Change"
        OnMouseUp: execute {
            IF active_param <> 0 THEN
            	active_param.Change_Param(value);
            	actual_value := active_param.display;
            END_IF
        }
    RoundedRectangle (20,80 300x50), "%s", text variable: name
END_VISUALIZATION

// ---- VISUs/LogVisu.TcVIS
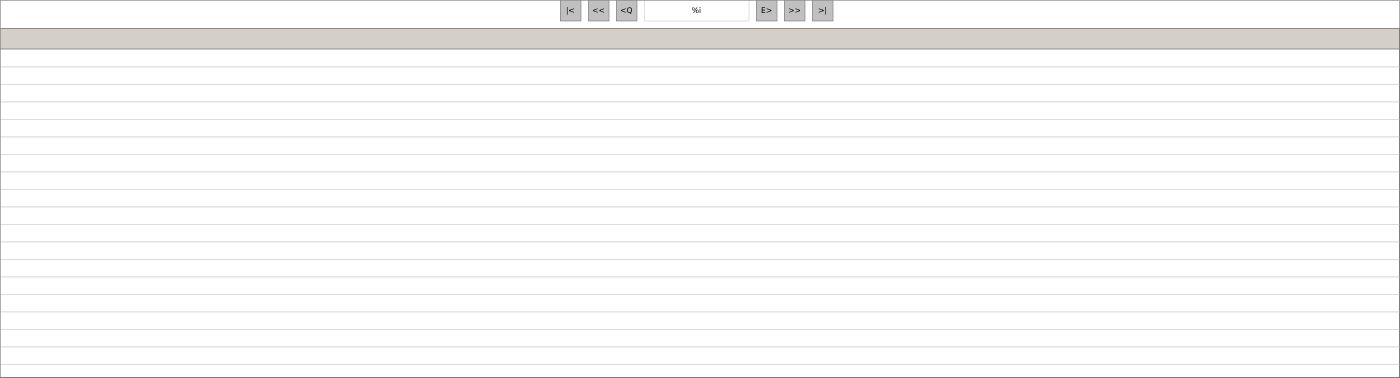
VISUALIZATION LogVisu  // 2000x540
VAR
	selected: INT := 1;
END_VAR
    Table (0,40 2000x500), data array: LogList.list
        p3854506369: LogList.list[INDEX]
        p1137915858: selected
    Textfield (920,0 150x30), "%i", text variable: selected
        OnMouseUp: write the text variable via Default, min 1
    RoundedRectangle (880,0 30x30), "<Q"
        OnMouseUp: execute {
            IF selected > 1 THEN
            	selected := selected - 1;
            END_IF
        }
    RoundedRectangle (1080,0 30x30), "E>"
        OnMouseUp: execute {
            IF selected < 4000 THEN
            	selected := selected + 1;
            END_IF
        }
    RoundedRectangle (840,0 30x30), "<<"
        OnMouseUp: execute {
            IF selected > 25 THEN
            	selected := selected - 24;
            END_IF
        }
    RoundedRectangle (1120,0 30x30), ">>"
        OnMouseUp: execute {
            IF selected < 3975 THEN
            	selected := selected + 24;
            END_IF
        }
    RoundedRectangle (800,0 30x30), "|<"
        OnMouseUp: execute { selected := 1; }
    RoundedRectangle (1160,0 30x30), ">|"
        OnMouseUp: execute { selected := LogList.lastlog; }
    hotkey HotkeyInput Id=481038434304, Key=KeyName=Q, VisuElemId=7
    hotkey HotkeyInput Id=481040531456, Key=KeyName=E, VisuElemId=18
END_VISUALIZATION
